(* PLC project SafeLOGIC-1, BrAutomation SafeDESIGNER  5.15.0.0 *)
(* stored: companyURL http://www.br-automation.com, creationDateTime Fri Jan 06 09:25:58 2023 *)

PROGRAM Main
  VAR  (* added by the conversion: wires and edge detectors of the diagram *)
    _OR260_OUT : BOOL;
    _AND_S274_OUT : ANY;
    _OR302_OUT : BOOL;
    _AND_S319_OUT : ANY;
    _AND_S350_OUT : ANY;
    _AND_S366_OUT : ANY;
  END_VAR

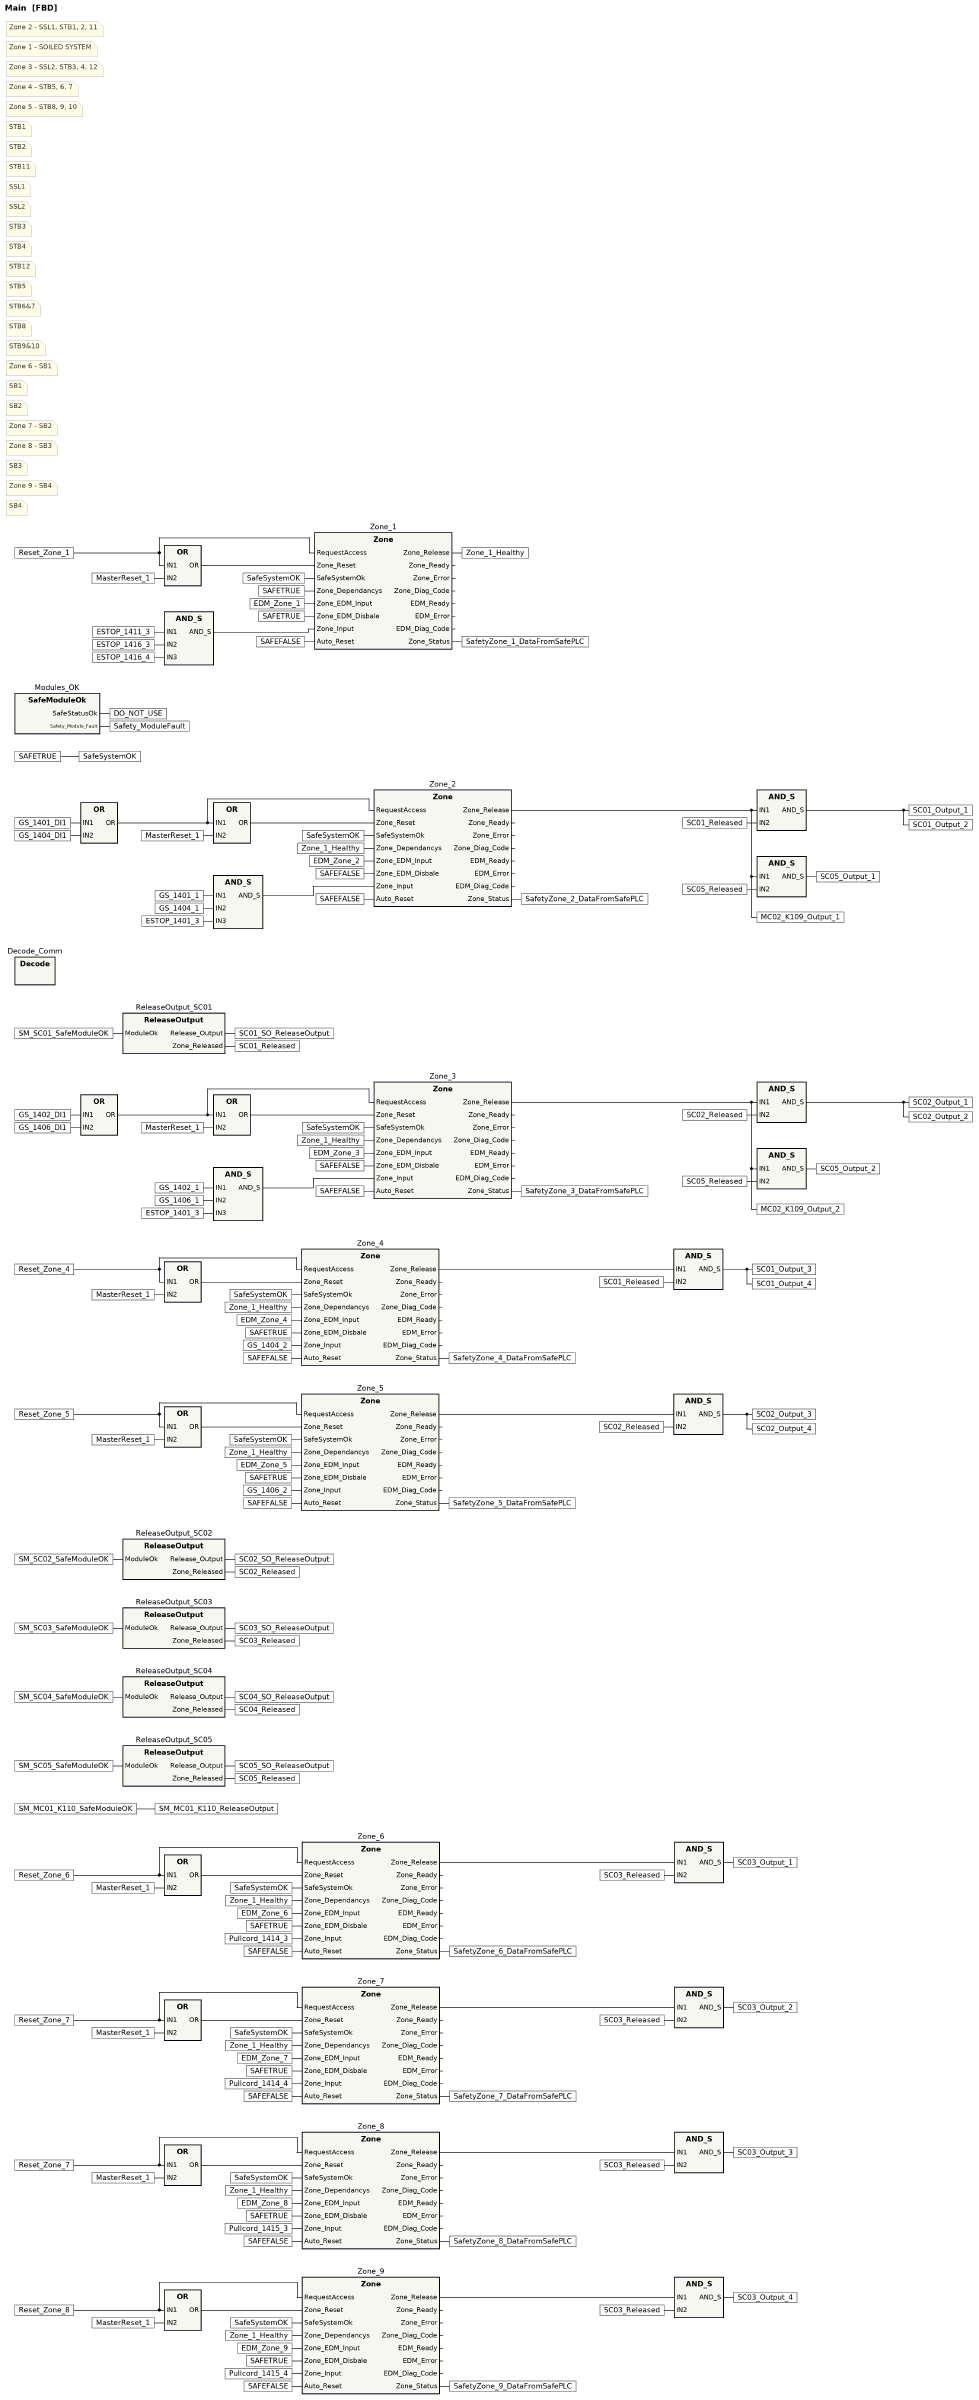
(* FBD diagram, written out as Structured Text *)
Modules_OK();
Safety_ModuleFault := Modules_OK.Safety_Module_Fault;
DO_NOT_USE := Modules_OK.SafeStatusOk;
SafeSystemOK := SAFETRUE;
SM_MC01_K110_ReleaseOutput := SM_MC01_K110_SafeModuleOK;
ReleaseOutput_SC01(ModuleOk := SM_SC01_SafeModuleOK);
SC01_Released := ReleaseOutput_SC01.Zone_Released;
SC01_SO_ReleaseOutput := ReleaseOutput_SC01.Release_Output;
ReleaseOutput_SC02(ModuleOk := SM_SC02_SafeModuleOK);
SC02_SO_ReleaseOutput := ReleaseOutput_SC02.Release_Output;
SC02_Released := ReleaseOutput_SC02.Zone_Released;
ReleaseOutput_SC03(ModuleOk := SM_SC03_SafeModuleOK);
SC03_SO_ReleaseOutput := ReleaseOutput_SC03.Release_Output;
SC03_Released := ReleaseOutput_SC03.Zone_Released;
ReleaseOutput_SC04(ModuleOk := SM_SC04_SafeModuleOK);
SC04_SO_ReleaseOutput := ReleaseOutput_SC04.Release_Output;
SC04_Released := ReleaseOutput_SC04.Zone_Released;
ReleaseOutput_SC05(ModuleOk := SM_SC05_SafeModuleOK);
SC05_SO_ReleaseOutput := ReleaseOutput_SC05.Release_Output;
SC05_Released := ReleaseOutput_SC05.Zone_Released;
(* Zone 1 - SOILED SYSTEM *)
Zone_1(RequestAccess := Reset_Zone_1, Zone_Reset := Reset_Zone_1 OR MasterReset_1, SafeSystemOk := SafeSystemOK, Zone_Dependancys := SAFETRUE, Zone_EDM_Input := EDM_Zone_1, Zone_EDM_Disbale := SAFETRUE, Zone_Input := AND_S(ESTOP_1411_3, ESTOP_1416_3, ESTOP_1416_4), Auto_Reset := SAFEFALSE);
Zone_1_Healthy := Zone_1.Zone_Release;
SafetyZone_1_DataFromSafePLC := Zone_1.Zone_Status;
(* Zone 2 - SSL1, STB1, 2, 11 *)
(* SSL1 *)
_OR260_OUT := GS_1401_DI1 OR GS_1404_DI1;
Zone_2(RequestAccess := _OR260_OUT, Zone_Reset := _OR260_OUT OR MasterReset_1, SafeSystemOk := SafeSystemOK, Zone_Dependancys := Zone_1_Healthy, Zone_EDM_Input := EDM_Zone_2, Zone_EDM_Disbale := SAFEFALSE, Zone_Input := AND_S(GS_1401_1, GS_1404_1, ESTOP_1401_3), Auto_Reset := SAFEFALSE);
MC02_K109_Output_1 := Zone_2.Zone_Release;
(* STB1 *)
(* STB2 *)
_AND_S274_OUT := AND_S(Zone_2.Zone_Release, SC01_Released);
SC01_Output_1 := _AND_S274_OUT;
SC01_Output_2 := _AND_S274_OUT;
(* STB11 *)
SafetyZone_2_DataFromSafePLC := Zone_2.Zone_Status;
SC05_Output_1 := AND_S(Zone_2.Zone_Release, SC05_Released);
(* Zone 3 - SSL2, STB3, 4, 12 *)
(* SSL2 *)
_OR302_OUT := GS_1402_DI1 OR GS_1406_DI1;
Zone_3(RequestAccess := _OR302_OUT, Zone_Reset := _OR302_OUT OR MasterReset_1, SafeSystemOk := SafeSystemOK, Zone_Dependancys := Zone_1_Healthy, Zone_EDM_Input := EDM_Zone_3, Zone_EDM_Disbale := SAFEFALSE, Zone_Input := AND_S(GS_1402_1, GS_1406_1, ESTOP_1401_3), Auto_Reset := SAFEFALSE);
MC02_K109_Output_2 := Zone_3.Zone_Release;
(* STB3 *)
(* STB4 *)
_AND_S319_OUT := AND_S(Zone_3.Zone_Release, SC02_Released);
SC02_Output_1 := _AND_S319_OUT;
SC02_Output_2 := _AND_S319_OUT;
(* STB12 *)
SafetyZone_3_DataFromSafePLC := Zone_3.Zone_Status;
SC05_Output_2 := AND_S(Zone_3.Zone_Release, SC05_Released);
(* Zone 4 - STB5, 6, 7 *)
(* STB5 *)
(* STB6&7 *)
Zone_4(RequestAccess := Reset_Zone_4, Zone_Reset := Reset_Zone_4 OR MasterReset_1, SafeSystemOk := SafeSystemOK, Zone_Dependancys := Zone_1_Healthy, Zone_EDM_Input := EDM_Zone_4, Zone_EDM_Disbale := SAFETRUE, Zone_Input := GS_1404_2, Auto_Reset := SAFEFALSE);
_AND_S350_OUT := AND_S(Zone_4.Zone_Release, SC01_Released);
SC01_Output_3 := _AND_S350_OUT;
SC01_Output_4 := _AND_S350_OUT;
SafetyZone_4_DataFromSafePLC := Zone_4.Zone_Status;
(* Zone 5 - STB8, 9, 10 *)
(* STB8 *)
(* STB9&10 *)
Zone_5(RequestAccess := Reset_Zone_5, Zone_Reset := Reset_Zone_5 OR MasterReset_1, SafeSystemOk := SafeSystemOK, Zone_Dependancys := Zone_1_Healthy, Zone_EDM_Input := EDM_Zone_5, Zone_EDM_Disbale := SAFETRUE, Zone_Input := GS_1406_2, Auto_Reset := SAFEFALSE);
_AND_S366_OUT := AND_S(Zone_5.Zone_Release, SC02_Released);
SC02_Output_3 := _AND_S366_OUT;
SC02_Output_4 := _AND_S366_OUT;
SafetyZone_5_DataFromSafePLC := Zone_5.Zone_Status;
(* Zone 6 - SB1 *)
(* SB1 *)
Zone_6(RequestAccess := Reset_Zone_6, Zone_Reset := Reset_Zone_6 OR MasterReset_1, SafeSystemOk := SafeSystemOK, Zone_Dependancys := Zone_1_Healthy, Zone_EDM_Input := EDM_Zone_6, Zone_EDM_Disbale := SAFETRUE, Zone_Input := Pullcord_1414_3, Auto_Reset := SAFEFALSE);
SC03_Output_1 := AND_S(Zone_6.Zone_Release, SC03_Released);
SafetyZone_6_DataFromSafePLC := Zone_6.Zone_Status;
(* Zone 7 - SB2 *)
(* SB2 *)
Zone_7(RequestAccess := Reset_Zone_7, Zone_Reset := Reset_Zone_7 OR MasterReset_1, SafeSystemOk := SafeSystemOK, Zone_Dependancys := Zone_1_Healthy, Zone_EDM_Input := EDM_Zone_7, Zone_EDM_Disbale := SAFETRUE, Zone_Input := Pullcord_1414_4, Auto_Reset := SAFEFALSE);
SC03_Output_2 := AND_S(Zone_7.Zone_Release, SC03_Released);
SafetyZone_7_DataFromSafePLC := Zone_7.Zone_Status;
(* Zone 8 - SB3 *)
(* SB3 *)
Zone_8(RequestAccess := Reset_Zone_7, Zone_Reset := Reset_Zone_7 OR MasterReset_1, SafeSystemOk := SafeSystemOK, Zone_Dependancys := Zone_1_Healthy, Zone_EDM_Input := EDM_Zone_8, Zone_EDM_Disbale := SAFETRUE, Zone_Input := Pullcord_1415_3, Auto_Reset := SAFEFALSE);
SC03_Output_3 := AND_S(Zone_8.Zone_Release, SC03_Released);
SafetyZone_8_DataFromSafePLC := Zone_8.Zone_Status;
(* Zone 9 - SB4 *)
(* SB4 *)
Zone_9(RequestAccess := Reset_Zone_8, Zone_Reset := Reset_Zone_8 OR MasterReset_1, SafeSystemOk := SafeSystemOK, Zone_Dependancys := Zone_1_Healthy, Zone_EDM_Input := EDM_Zone_9, Zone_EDM_Disbale := SAFETRUE, Zone_Input := Pullcord_1415_4, Auto_Reset := SAFEFALSE);
SC03_Output_4 := AND_S(Zone_9.Zone_Release, SC03_Released);
SafetyZone_9_DataFromSafePLC := Zone_9.Zone_Status;
Decode_Comm();
END_PROGRAM
